{attribute 'OPC.UA.DA' := '1'}
FUNCTION_BLOCK SJH108Ionizer EXTENDS IonizerBase
VAR_INPUT
	
END_VAR
VAR_OUTPUT
END_VAR
VAR
	{attribute 'OPC.UA.DA' := '0'}
	_config : SJH108IonizerConfig;	
	{attribute 'OPC.UA.DA' := '0'}
	IoSJH108A : IoSJH108A;
	
	{attribute 'OPC.UA.DA' := '0'}
	_initDevice : BOOL;	
	
	{region 'Commands'}	
		 	
	{attribute 'OPC.UA.DA' := '0'}
	_openAirValveCmd : BOOL;	
	{attribute 'OPC.UA.DA' := '0'}
	_openValve : BOOL;
	{attribute 'OPC.UA.DA' := '0'}
	_enableStaticEliminationInterruptCmd : BOOL;
	{attribute 'OPC.UA.DA' := '0'}
	_enable : BOOL;
	{attribute 'OPC.UA.DA' := '0'}			  		   
	_raisePropertiesCmd : BOOL;	 
			
	{endregion}		 
	
	{attribute 'OPC.UA.DA' := '0'}
	_deliverMessages : INT;	
		 	
	AlarmMsg : STRING(255);
	AirValveIsOpenMsg : STRING(255);
	StaticEliminationInterruptMsg : STRING(255);
	RefreshingMsg : STRING(255);
	
	{attribute 'OPC.UA.DA' := '0'}
	message : STRING;
	
	{attribute 'OPC.UA.DA' := '0'}
	_itemScheduler : INT;
	{attribute 'OPC.UA.DA' := '0'}
	_itemRaisedProperties : INT;			
	{attribute 'OPC.UA.DA' := '0'}
	_pulseGenerator : TON;	
	
	{attribute 'OPC.UA.DA' := '0'}
	tmpConcat1 : STRING;
	{attribute 'OPC.UA.DA' := '0'}
	tmpConcat2 : STRING;
	{attribute 'OPC.UA.DA' := '0'}
	tmpConcatName : STRING; 
	{attribute 'OPC.UA.DA' := '0'}
	tmpConcatDescription : STRING;
	{attribute 'OPC.UA.DA' := '0'}
	tmpConcatAlarmID : STRING;	
	{attribute 'OPC.UA.DA' := '0'}
	_alarmCount : UINT;
	
	
END_VAR

SUPER^();

// Init device
InitDevice();

CASE _deliverMessages OF	
	EFeedbackMsgSJH108.AlarmMsg :
		AlarmMsg := message;
	EFeedbackMsgSJH108.AirValveIsOpenMsg :
		AirValveIsOpenMsg := TO_STRING(IoSJH108A.OutputOpenAirValve);
END_CASE
		
// Commands		
OpensAirValve(_openAirValveCmd, _openValve);
EnableStaticEliminationInterrupt(_enableStaticEliminationInterruptCmd, _enable);
RaisePropertiesChanged(_raisePropertiesCmd);

IF (NOT _openAirValveCmd AND NOT _enableStaticEliminationInterruptCmd AND NOT _raisePropertiesCmd) THEN	
	MessageScheduler();
END_IF

{attribute 'TcRpcEnable' := '1'}
METHOD PRIVATE EnableStaticEliminationInterrupt
VAR_INPUT
	Execute : BOOL;
	Enable : BOOL;
END_VAR
IF Execute THEN		
	_enable := Enable;
	_logger.Information(_message.Reset().Append(_config.Name).Append(' - EnableStaticEliminationInterrupt=').Append(TO_STRING(_enable)).ToString());
		
	IoSJH108A.OutputStaticEliminationInterrupt := _enable;
	_enableStaticEliminationInterruptCmd := FALSE;		
END_IF
END_METHOD

METHOD FB_init : BOOL
VAR_INPUT
	bInitRetains : BOOL; // if TRUE, the retain variables are initialized (warm start / cold start)
	bInCopyCode : BOOL;  // if TRUE, the instance afterwards gets moved into the copy code (online change)
	Config : SJH108IonizerConfig;
END_VAR
IF Config.IsEnabled THEN
	_config := Config;
	
	SUPER^._ionizerConfig.Name := Config.Name;
	SUPER^._ionizerConfig.DeviceID := Config.DeviceID;
	SUPER^._ionizerConfig.IsEnabled := Config.IsEnabled;
	SUPER^._ionizerConfig.LogLevel := Config.LogLevel;
	
	SUPER^.Name := Config.Name;
	SUPER^.DeviceID := Config.DeviceID;	
	THIS^.Family := DeviceFamily.Ionizer;
		
	IoSJH108A.OutputOpenAirValve := TRUE;
	
	_Logger.Information(_message.Reset().Append('Init ').
							Append('{').Append(TO_STRING(THIS^.Family)).Append('} - ').
							Append('{').Append(TO_STRING(Config.Name)).Append('}').ToString());																													
END_IF
END_METHOD

METHOD InitDevice
VAR_INPUT
END_VAR
IF NOT _initDevice THEN	
	_logger.Information(_message.Reset().Append(_config.Name).Append(' - Init device').ToString());
	
	THIS^.SetDone();	
	_initDevice := TRUE;	
END_IF
END_METHOD

METHOD MessageScheduler
VAR_INPUT
END_VAR
IF _pulseGenerator.Q THEN
	_pulseGenerator(IN := FALSE, PT := T#10MS);
	
	message := ' ';
	CASE _itemScheduler OF			
		0:  AirValveIsOpenMsg := ' ';
			_itemScheduler := 1;
			
		1:	ReadAlarm(); 
			_itemScheduler := 0;
	END_CASE
ELSE
	_pulseGenerator(IN := TRUE, PT := T#100MS);		
END_IF
END_METHOD

{attribute 'TcRpcEnable' := '1'}
METHOD PRIVATE OpensAirValve
VAR_INPUT
	Execute : BOOL;
	OpenValve : BOOL;
END_VAR
IF Execute THEN	
	_openValve := OpenValve;	
	_logger.Information(_message.Reset().Append(_config.Name).Append(' - Open=').Append(TO_STRING(_openValve)).ToString());
	
	IoSJH108A.OutputOpenAirValve := _openValve;
	
	_openAirValveCmd := FALSE;		
END_IF
END_METHOD

{attribute 'TcRpcEnable' := '1'}
METHOD RaisePropertiesChanged
VAR_INPUT
	Execute : BOOL;
END_VAR
IF Execute THEN		
	_raisePropertiesCmd := TRUE;	
	
	IF _pulseGenerator.Q THEN
		_pulseGenerator(IN := FALSE, PT := T#10MS);
		
		CASE _itemRaisedProperties OF		
			0:  RefreshingMsg := TO_STRING(TRUE);
				_alarmCount := 0;
				_itemRaisedProperties := 1;
				
			1: 	ReadAlarm();
				_alarmCount := _alarmCount + 1;
				IF _alarmCount = IonizerConst.NUMBER_ALARMS THEN
					_itemRaisedProperties := 2;
				END_IF							
			
			2:  RefreshingMsg := TO_STRING(FALSE);
				_raisePropertiesCmd := FALSE;
				_itemRaisedProperties := 0;		
		END_CASE	
	ELSE
		_pulseGenerator(IN := TRUE, PT := T#100MS);	
	END_IF
END_IF
END_METHOD

METHOD ReadAlarm
VAR_INPUT
END_VAR
VAR
	triggered : BOOL;
END_VAR
_deliverMessages := EFeedbackMsgSJH108.AlarmMsg;

_alarmCount := 0;

tmpConcatName := CONCAT(_config.IonizerAlarm[_alarmCount].Name, ';');
tmpConcatDescription := CONCAT(_config.IonizerAlarm[_alarmCount].Description, ';');
tmpConcatAlarmID := CONCAT(UINT_TO_STRING(_config.IonizerAlarm[_alarmCount].AlarmID), ';');

tmpConcat1 := CONCAT(tmpConcatName, tmpConcatDescription);
tmpConcat2 := CONCAT(tmpConcat1, tmpConcatAlarmID);

IF _config.IonizerAlarm[_alarmCount].Triggered THEN
	triggered := FALSE;
ELSE
	triggered := TRUE;
END_IF

message := CONCAT(tmpConcat2, TO_STRING(triggered));
END_METHOD

END_FUNCTION_BLOCK

(* stored: Version 1.1.0.1, ProductVersion 3.1.4024.12
   POU SJH108Ionizer: Id {877406b8-0bd3-490a-a6af-0813a8d62411}, SpecialFunc None
   Folder Commands: Id {bd3ddf92-3ebd-457e-9c68-037f07551c70}
   Method EnableStaticEliminationInterrupt: Id {01c5c83f-779b-46f5-b75a-ead75412fb71}
   Method FB_init: Id {c4f9e8ae-dc45-470f-b179-ac7ece289020}
   Method InitDevice: Id {d7d2e8d7-3700-45d6-8253-8e742150dd1f}
   Method MessageScheduler: Id {24666361-8eb1-4866-8a5e-11e47ab2eb59}
   Method OpensAirValve: Id {2fb73b5e-e5bf-4037-844a-f9c5a1431a1a}
   Method RaisePropertiesChanged: Id {7df441c7-aee6-41eb-a3c6-a70217d04ad2}
   Method ReadAlarm: Id {2a0071be-c731-4d1e-914f-b5e0fa5bb30f} *)
